TYPE ST_Empty :
STRUCT
	{attribute 'hide'}
	BUnknown						: BYTE;
	BState							: BYTE;
(* wDiagnosis *)
	{attribute 'hide'}
	bDiagBIT0						: BIT; 		(* Empty *)
	{attribute 'hide'}
	bDiagBIT1						: BIT; 		(* Empty *)
	{attribute 'hide'}
	bDiagBIT2						: BIT; 		(* Empty *)
	{attribute 'hide'}
	bDiagBIT3						: BIT; 		(* Empty *)
	{attribute 'hide'}
	bDiagBIT4						: BIT; 		(* Empty *)
	{attribute 'hide'}
	bDiagBIT5						: BIT; 		(* Empty *)
	{attribute 'hide'}
	bDiagBIT6						: BIT; 		(* Empty *)
	{attribute 'hide'}
	bDiagBIT7						: BIT; 		(* Empty *)
	{attribute 'hide'}
	bDiagBIT8						: BIT; 		(* Empty *)
	{attribute 'hide'}
	bDiagBIT9						: BIT; 		(* Empty *)
	{attribute 'hide'}
	bDiagBIT10						: BIT; 		(* Empty *)
	{attribute 'hide'}
	bDiagBIT11						: BIT; 		(* Empty *)
	{attribute 'hide'}
	bDiagBIT12						: BIT; 		(* Empty *)
	{attribute 'hide'}
	bDiagBIT13						: BIT; 		(* Empty *)
	{attribute 'hide'}
	bDiagBIT14						: BIT; 		(* Empty *)
	{attribute 'hide'}
	bDiagBIT15						: BIT; 		(* Empty *)
(* wInputs *)
	{attribute 'hide'}
	bInputBIT0						: BIT; 		(* Empty *)
	{attribute 'hide'}
	bInputBIT1						: BIT; 		(* Empty *)
	{attribute 'hide'}
	bInputBIT2						: BIT; 		(* Empty *)
	{attribute 'hide'}
	bInputBIT3						: BIT; 		(* Empty *)
	{attribute 'hide'}
	bInputBIT4						: BIT; 		(* Empty *)
	{attribute 'hide'}
	bInputBIT5						: BIT; 		(* Empty *)
	{attribute 'hide'}
	bInputBIT6						: BIT; 		(* Empty *)
	{attribute 'hide'}
	bInputBIT7						: BIT; 		(* Empty *)
	{attribute 'hide'}
	bInputBIT8						: BIT; 		(* Empty *)
	{attribute 'hide'}
	bInputBIT9						: BIT; 		(* Empty *)
	{attribute 'hide'}
	bInputBIT10						: BIT; 		(* Empty *)
	{attribute 'hide'}
	bInputBIT11						: BIT; 		(* Empty *)
	{attribute 'hide'}
	bInputBIT12						: BIT; 		(* Empty *)
	{attribute 'hide'}
	bInputBIT13						: BIT; 		(* Empty *)
	{attribute 'hide'}
	bInputBIT14						: BIT; 		(* Empty *)
	{attribute 'hide'}
	bInputBIT15						: BIT; 		(* Empty *)
(* wOutputs *)
	{attribute 'hide'}
	bOutputBIT0						: BIT; 		(* Empty *)
	{attribute 'hide'}
	bOutputBIT1						: BIT; 		(* Empty *)
	{attribute 'hide'}
	bOutputBIT2						: BIT; 		(* Empty *)
	{attribute 'hide'}
	bOutputBIT3						: BIT; 		(* Empty *)
	{attribute 'hide'}
	bOutputBIT4						: BIT; 		(* Empty *)
	{attribute 'hide'}
	bOutputBIT5						: BIT; 		(* Empty *)
	{attribute 'hide'}
	bOutputBIT6						: BIT; 		(* Empty *)
	{attribute 'hide'}
	bOutputBIT7						: BIT; 		(* Empty *)
	{attribute 'hide'}
	bOutputBIT8						: BIT; 		(* Empty *)
	{attribute 'hide'}
	bOutputBIT9						: BIT; 		(* Empty *)
	{attribute 'hide'}
	bOutputBIT10					: BIT; 		(* Empty *)
	{attribute 'hide'}
	bOutputBIT11					: BIT; 		(* Empty *)
	{attribute 'hide'}
	bOutputBIT12					: BIT; 		(* Empty *)
	{attribute 'hide'}
	bOutputBIT13					: BIT; 		(* Empty *)
	{attribute 'hide'}
	bOutputBIT14					: BIT; 		(* Empty *)
	{attribute 'hide'}
	bOutputBIT15					: BIT; 		(* Empty *)
END_STRUCT
END_TYPE

(* stored: Version 1.1.0.1, ProductVersion 3.1.4022.12
   DUT ST_Empty: Id {e0e945c8-b7c4-46d9-b101-822f3e1ba6c9} *)
